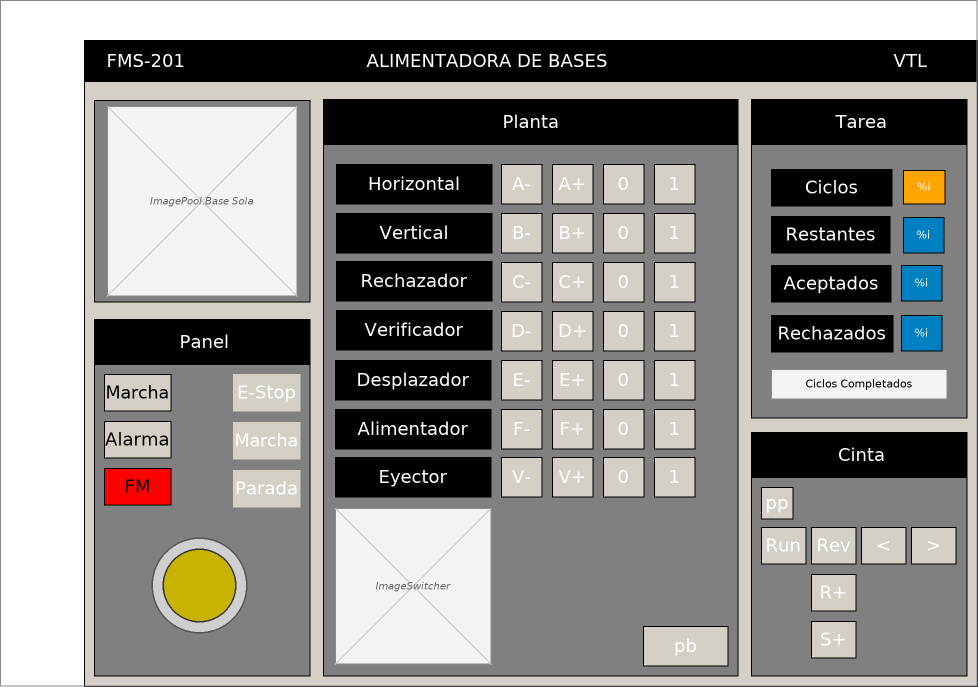
VISUALIZATION Visualization  // 978x687
    Rectangle (84,81 894x606)
    Rectangle (751,144 216x274)
    Rectangle (323,144 415x532)
    Rectangle (323,99 415x45)
    Label (323,101 416x42), "Planta"
    Rectangle (751,99 216x45)
    Label (801,104 121x36), "Tarea"
    Progressbar (771,369 176x30), "Ciclos Completados", variable: MAIN.test_pieza.Aceptados
    RoundedRectangle (336,164 156x40), "Horizontal", colour toggle: MAIN.test_pieza.Descargador_adelante
    Textfield (903,170 42x34), "%i", text variable: MAIN.test_pieza.Ciclos
        OnMouseDown: write MAIN.test_pieza.Ciclos via VisuDialogs.Numpad, min 1, max 10
    RoundedRectangle (771,169 121x37), "Ciclos"
    RoundedRectangle (771,216 119x37), "Restantes"
    RoundedRectangle (771,265 120x37), "Aceptados"
    RoundedRectangle (771,315 122x37), "Rechazados"
    Textfield (903,217 41x36), "%i", text variable: MAIN.test_pieza.Restantes
    Textfield (901,265 41x36), "%i", text variable: MAIN.test_pieza.Aceptados
    Textfield (901,315 41x36), "%i", text variable: MAIN.test_pieza.Rechazados
    RoundedRectangle (552,213 41x40), "B+", colour toggle: MAIN.test_pieza.Descargador_baja
        toggle MAIN.test_pieza.Descargador_baja
    Rectangle (751,477 216x199)
    Rectangle (751,432 216x45)
    Label (801,437 121x36), "Cinta"
    Rectangle (94,100 216x202)
    Rectangle (94,364 216x312)
    Rectangle (94,319 216x45)
    Label (144,324 121x36), "Panel"
    Rectangle (84,40 894x41)
    Label (84,41 893x40), "FMS-201 ALIMENTADORA DE BASES VTL"
    RoundedRectangle (336,213 156x40), "Vertical", colour toggle: MAIN.test_pieza.Descargador_adelante
    RoundedRectangle (552,164 41x40), "A+", colour toggle: MAIN.test_pieza.Descargador_adelante
        tap MAIN.test_pieza.Descargador_adelante
    RoundedRectangle (552,262 41x40), "C+", colour toggle: MAIN.test_pieza.Rechazador_adelante
        tap MAIN.test_pieza.Rechazador_adelante
    RoundedRectangle (552,311 41x40), "D+", colour toggle: MAIN.test_pieza.Verificador_baja
        tap MAIN.test_pieza.Verificador_baja
    RoundedRectangle (552,360 41x40), "E+", colour toggle: MAIN.test_pieza.Desplazador_adelante
        tap MAIN.test_pieza.Desplazador_adelante
    RoundedRectangle (552,409 41x40), "F+", colour toggle: MAIN.test_pieza.Alimentador_adelante
        tap MAIN.test_pieza.Alimentador_adelante
        toggle MAIN.test_pieza.Descargador_baja
    RoundedRectangle (552,457 41x40), "V+", colour toggle: MAIN.test_pieza.Eyector_succiona
        toggle MAIN.test_pieza.Eyector_succiona
    RoundedRectangle (336,261 156x40), "Rechazador", colour toggle: MAIN.test_pieza.Descargador_adelante
    RoundedRectangle (336,310 156x40), "Verificador", colour toggle: MAIN.test_pieza.Descargador_adelante
    RoundedRectangle (335,360 156x40), "Desplazador", colour toggle: MAIN.test_pieza.Descargador_adelante
    RoundedRectangle (335,409 156x40), "Alimentador", colour toggle: MAIN.test_pieza.Descargador_adelante
    RoundedRectangle (335,457 156x40), "Eyector", colour toggle: MAIN.test_pieza.Descargador_adelante
    RoundedRectangle (501,164 41x40), "A-", colour toggle: MAIN.test_pieza.Descargador_atras
        tap MAIN.test_pieza.Descargador_atras
    RoundedRectangle (603,164 41x40), "0", colour toggle: MAIN.test_pieza.Horizontal_descargador_detras
        tap MAIN.test_pieza.Horizontal_descargador_detras
    RoundedRectangle (654,164 41x40), "1", colour toggle: MAIN.test_pieza.Horizontal_descargador_delante
        tap MAIN.test_pieza.Horizontal_descargador_delante
    RoundedRectangle (603,213 41x40), "0", colour toggle: MAIN.test_pieza.Vertical_descargador_arriba
        tap MAIN.test_pieza.Vertical_descargador_arriba
    RoundedRectangle (654,213 41x40), "1", colour toggle: MAIN.test_pieza.Vertical_descargador_abajo
        tap MAIN.test_pieza.Vertical_descargador_abajo
    RoundedRectangle (603,262 41x40), "0"
    RoundedRectangle (603,311 41x40), "0", colour toggle: MAIN.test_pieza.Verificador_arriba
        tap MAIN.test_pieza.Verificador_arriba
    RoundedRectangle (603,360 41x40), "0", colour toggle: MAIN.test_pieza.Desplazador_detras
        tap MAIN.test_pieza.Desplazador_detras
    RoundedRectangle (603,409 41x40), "0", colour toggle: MAIN.test_pieza.Alimentador_detras
        tap MAIN.test_pieza.Alimentador_detras
    RoundedRectangle (603,457 41x40), "0"
    RoundedRectangle (654,262 41x40), "1"
    RoundedRectangle (654,311 41x40), "1", colour toggle: MAIN.test_pieza.Verificador_abajo
        tap MAIN.test_pieza.Verificador_abajo
    RoundedRectangle (654,360 41x40), "1"
    RoundedRectangle (654,409 41x40), "1", colour toggle: MAIN.test_pieza.Alimentador_delante
        tap MAIN.test_pieza.Alimentador_delante
    RoundedRectangle (654,457 41x40), "1", colour toggle: MAIN.test_pieza.Vacio_obtenido_vacuostato_descargador
        tap MAIN.test_pieza.Vacio_obtenido_vacuostato_descargador
    RoundedRectangle (501,213 41x40), "B-"
    RoundedRectangle (501,262 41x40), "C-"
    RoundedRectangle (501,311 41x40), "D-"
    RoundedRectangle (501,360 41x40), "E-"
    RoundedRectangle (501,409 41x40), "F-"
    RoundedRectangle (501,457 41x40), "V-"
    RoundedRectangle (643,626 85x40), "pb", colour toggle: MAIN.test_pieza.Base_en_Alimentador
        tap MAIN.test_pieza.Base_en_Alimentador
    RoundedRectangle (104,468 67x37), "FM", colour toggle: MAIN.test_pieza.Lampara_falta_material
        tap MAIN.test_pieza.Lampara_falta_material
    RoundedRectangle (761,487 32x32), "pp", colour toggle: MAIN.test_pieza.Presencia_pale
        tap MAIN.test_pieza.Presencia_pale
    RoundedRectangle (911,527 45x37), ">", colour toggle: MAIN.test_pieza.Activa_marcha_motor_cinta
        tap MAIN.test_pieza.Activa_marcha_motor_cinta
    RoundedRectangle (861,527 45x37), "<", colour toggle: MAIN.test_pieza.Invierte_marcha_motor_cinta
        toggle MAIN.test_pieza.Invierte_marcha_motor_cinta
    RoundedRectangle (761,527 45x37), "Run", colour toggle: MAIN.test_pieza.Activa_marcha_motor_cinta
    RoundedRectangle (811,527 45x37), "Rev", colour toggle: MAIN.test_pieza.Invierte_marcha_motor_cinta
    RoundedRectangle (811,574 45x37), "R+", colour toggle: MAIN.test_pieza.Retenedor_pale_baja
        tap MAIN.test_pieza.Retenedor_pale_baja
    RoundedRectangle (811,621 45x37), "S+", colour toggle: MAIN.test_pieza.Separador_pale_sube
        tap MAIN.test_pieza.Separador_pale_sube
    RoundedRectangle (233,374 67x37), "E-Stop", colour toggle: MAIN.test_pieza.Pulsador_parada_emergencia
        tap MAIN.test_pieza.Pulsador_parada_emergencia
    RoundedRectangle (233,422 67x37), "Marcha", colour toggle: MAIN.test_pieza.Pulsador_marcha
        tap MAIN.test_pieza.Pulsador_marcha
    RoundedRectangle (233,470 67x37), "Parada", colour toggle: MAIN.test_pieza.Pulsador_parada_NC
        tap MAIN.test_pieza.Pulsador_parada_NC
    RoundedRectangle (104,421 67x37), "Alarma", colour toggle: MAIN.test_pieza.Lampara_alarma
        tap MAIN.test_pieza.Lampara_alarma
    RoundedRectangle (104,374 67x37), "Marcha", colour toggle: MAIN.test_pieza.Lampara_marcha
        tap MAIN.test_pieza.Lampara_marcha
    Image (107,106 190x190), image: ImagePool.Base Sola
    Lamp1 (142,530 115x111), variable: MAIN.test_pieza.Lampara_falta_material, style: Lamp-Lamp1-Yellow
    ImageSwitcher (335,508 156x156), variable: MAIN.test_pieza.pieza_ok, background image: ImagePool.Base OK, image: ImagePool.Base No OK, behaviour: TOGGLE
END_VISUALIZATION

(* stored: Version 1.1.0.1, ProductVersion 3.1.4024.12
   Visu Visualization: Id {d064ae99-b9a1-47bf-8163-5ceaadee03a3} *)
